FUNCTION_BLOCK ABSTRACT FB_AbstractObservable EXTENDS FB_Object IMPLEMENTS I_Observable
VAR
    // Attributes
    _nTypeClass:                __SYSTEM.TYPE_CLASS;
    _bAutoNotify:               BOOL := TRUE; // Notify automatically on write access of observable value
    _bNotifyWhenChanged:        BOOL; // Notify only when the value is actually changed

    // Dynamic mem
    _fbObsList:                 FB_List; // Observer list

    _fbNotifyObservers:         FB_NotifyObserverAction;
END_VAR

METHOD Attach : BOOL
VAR_INPUT
    ipObserver:     I_Observer;
END_VAR
IF ipObserver = 0 // Invalid interface pointer
    OR_ELSE ipObserver.nTypeClass <> THIS^._nTypeClass // Invalid type
    OR_ELSE THIS^.Contains(ipObserver) // Already added
    THEN
    RETURN;
END_IF

Attach := THIS^._fbObsList.AddItem(ipObserver) <> -1;

IF Attach THEN
    THIS^.NotifyLast();
END_IF
END_METHOD

(*Notify automatically on write access of observable value*)
PROPERTY bAutoNotify : BOOL
GET
bAutoNotify := THIS^._bAutoNotify;
END_GET
SET
THIS^._bAutoNotify := bAutoNotify;
END_SET
END_PROPERTY

PROPERTY bNotifyWhenChanged : BOOL
GET
bNotifyWhenChanged := THIS^._bNotifyWhenChanged;
END_GET
SET
THIS^._bNotifyWhenChanged := bNotifyWhenChanged;
END_SET
END_PROPERTY

METHOD ClearAll
VAR_INPUT
END_VAR
THIS^._fbObsList.Clear();
END_METHOD

METHOD Contains : BOOL
VAR_INPUT
    ipObserver: I_Observer;
END_VAR
Contains := THIS^._fbObsList.Contains(ipObserver);
END_METHOD

METHOD Detach : BOOL
VAR_INPUT
    ipObserver:     I_Observer;
END_VAR
Detach := THIS^._fbObsList.Remove(ipObserver);
END_METHOD

PROPERTY ABSTRACT nDataSize : UDINT
GET
END_GET
END_PROPERTY

PROPERTY nObserverCount : UDINT
GET
nObserverCount := THIS^._fbObsList.nCount;
END_GET
END_PROPERTY

METHOD NotifyAll : I_Observable
NotifyAll := THIS^;

THIS^._fbObsList.ForEach(
    THIS^._fbNotifyObservers
         .Inputs(THIS^.pData,
                 THIS^._nTypeClass,
                 THIS^.nDataSize));
END_METHOD

METHOD NotifyLast : I_Observable
VAR
    ipLastObs: I_Observer;
END_VAR
NotifyLast := THIS^;

ipLastObs := THIS^.ObserverAt(TO_DINT(THIS^.nObserverCount) - 1);

IF ipLastObs <> 0 THEN
    ipLastObs.UpdateP(pData := THIS^.pData,
                      nTypeClass := THIS^._nTypeClass,
                      nSize := THIS^.nDataSize);
END_IF
END_METHOD

METHOD PROTECTED NotifyWithConditions : I_Observable
VAR_INPUT
END_VAR
NotifyWithConditions := THIS^;

IF NOT THIS^._bAutoNotify THEN
    RETURN;
END_IF

IF THIS^._bNotifyWhenChanged
    AND_THEN NOT THIS^.ValueChanged() THEN
    RETURN;
END_IF

THIS^.NotifyAll();
END_METHOD

PROPERTY nTypeClass : __SYSTEM.TYPE_CLASS
GET
nTypeClass := THIS^._nTypeClass;
END_GET
END_PROPERTY

METHOD ObserverAt : I_Observer
VAR_INPUT
    nIdx: DINT;
END_VAR
__QUERYINTERFACE(THIS^._fbObsList.ItemAt(nIdx), ObserverAt);
END_METHOD

PROPERTY PROTECTED ABSTRACT pData : POINTER TO BYTE
GET
END_GET
END_PROPERTY

METHOD ABSTRACT ValueChanged : BOOL
VAR_INPUT
END_VAR
END_METHOD

END_FUNCTION_BLOCK

(* stored: Version 1.1.0.1, ProductVersion 3.1.4024.12
   POU FB_AbstractObservable: Id {71e23688-66a9-4733-83ac-d64ef266e10a}, SpecialFunc None
   Method Attach: Id {2d2b36e2-7095-4ca4-b111-9d7fc9cde5fd}
   Property bAutoNotify: Id {74df07db-08be-0573-3a37-5dccf1e7dd5d}
   Get Get: Id {a06b71cf-b5b1-0175-3fce-b660054066b7}
   Set Set: Id {f620f6a5-c227-0747-3833-7da8408dde07}
   Property bNotifyWhenChanged: Id {fa76d4ca-250f-06a1-1b4a-98443338ae81}
   Get Get: Id {a9c32db7-d8ca-0b27-2cec-3449b9ed6a56}
   Set Set: Id {3bd698f8-1830-0ba9-1433-e88070376d5d}
   Method ClearAll: Id {d2ff27ca-2474-076b-3175-e48fff67c7aa}
   Method Contains: Id {76aabba0-b9ac-01e9-0b01-8a8b30e6a647}
   Method Detach: Id {cd87a177-86aa-454f-9754-8649faed008d}
   Property nDataSize: Id {06add94f-024a-47dc-87bf-b64b73b81f23}
   Get Get: Id {0f065d40-3079-435c-abd4-35bc9982957a}
   Property nObserverCount: Id {8a1f52c0-3800-483e-a595-61cd3c373210}
   Get Get: Id {11fffc9e-f7b8-44c7-97d9-9f9f0d9e2267}
   Method NotifyAll: Id {50b7b6ea-de79-46bd-bf28-05ba956e9a25}
   Method NotifyLast: Id {bfb98185-9d2f-403d-8101-4e4bed875c91}
   Method NotifyWithConditions: Id {b742a386-1bb7-051d-3dff-2af66164d0e9}
   Property nTypeClass: Id {1858b07f-e893-0a1d-310c-1f93f7d39211}
   Get Get: Id {ee9d73be-04be-0396-0ea3-61aae24b72b3}
   Method ObserverAt: Id {b9e320b9-08ab-450b-b4c7-7a324f7bf6f8}
   Property pData: Id {dc2c7af6-7d54-4c13-8681-c25bac9e7fcb}
   Get Get: Id {13c43774-fcc5-43db-b9fd-56325378b403}
   Method ValueChanged: Id {010c3d67-bfde-02a5-1223-efc7d35699a5} *)
